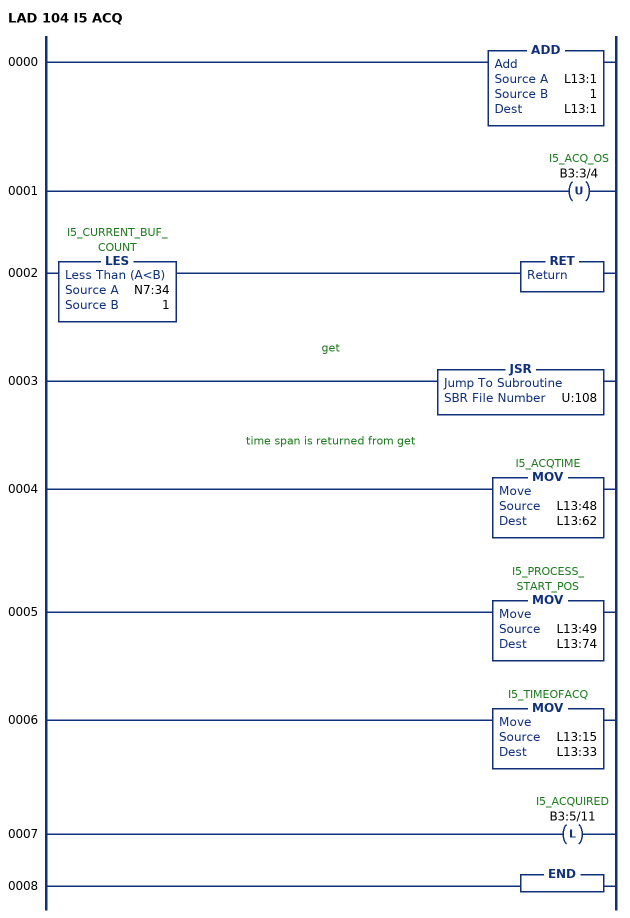
% Rung: 0 %
SOR ADD L13:1 1 L13:1 EOR
% Rung: 1 %
SOR OTU B3:3/4 EOR
%   B3:3/4  I5_ACQ_OS %
% Rung: 2 %
SOR LES N7:34 1 RET EOR
%   N7:34  I5_CURRENT_BUF_COUNT %
% Rung: 3 %
% get %
SOR JSR U:108 EOR
% Rung: 4 %
% time span is returned from get %
SOR MOV L13:48 L13:62 EOR
%   L13:48  I5_TIME_SPAN %
%   L13:62  I5_ACQTIME %
% Rung: 5 %
SOR MOV L13:49 L13:74 EOR
%   L13:49  I5_PULLED_POSITION %
%   L13:74  I5_PROCESS_START_POS %
% Rung: 6 %
SOR MOV L13:15 L13:33 EOR
%   L13:15  THE_TIME %
%   L13:33  I5_TIMEOFACQ %
% Rung: 7 %
SOR OTL B3:5/11 EOR
%   B3:5/11  I5_ACQUIRED %
% Rung: 8 %
SOR END EOR

LADDER 105 "I5 TESTER"
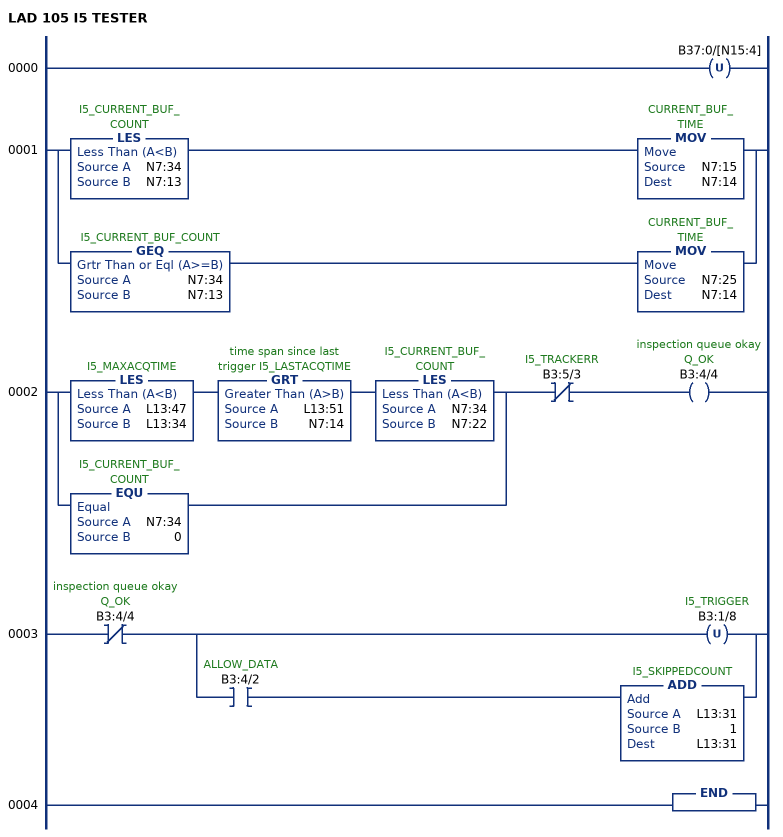
% Rung: 0 %
SOR OTU B37:0/[N15:4] EOR
%   B37:0  TOPGOOD1 %
%   N15:4  I5_TRIG_LOC %
% Rung: 1 %
SOR BST LES N7:34 N7:13 MOV N7:15 N7:14 NXB GEQ N7:34 N7:13 MOV N7:25 N7:14 BND EOR
%   N7:34  I5_CURRENT_BUF_COUNT %
%   N7:13  BUF_TRANS  "cam to pc buf transition" %
%   N7:15  CAM_BUF_TIME  "cam buf time" %
%   N7:14  CURRENT_BUF_TIME %
%   N7:25  PC_BUF_TIME  "pc buf time" %
% Rung: 2 %
SOR BST LES L13:47 L13:34 GRT L13:51 N7:14 LES N7:34 N7:22 NXB EQU N7:34 0 BND XIO B3:5/3 OTE B3:4/4 EOR
%   L13:47  I5_MAXACQTIME %
%   L13:34  MAX_ACQ_ALL  "absolute max acquire time before bypass trigger" %
%   L13:51  I5_LASTACQTIME  "time span since last trigger" %
%   N7:14  CURRENT_BUF_TIME %
%   N7:34  I5_CURRENT_BUF_COUNT %
%   N7:22  MAX_BUF_ALL  "max buffer count alowed before bypass" %
%   B3:5/3  I5_TRACKERR %
%   B3:4/4  Q_OK  "inspection queue okay" %
% Rung: 3 %
SOR XIO B3:4/4 BST OTU B3:1/8 NXB XIC B3:4/2 ADD L13:31 1 L13:31 BND EOR
%   B3:4/4  Q_OK  "inspection queue okay" %
%   B3:1/8  I5_TRIGGER %
%   B3:4/2  ALLOW_DATA %
%   L13:31  I5_SKIPPEDCOUNT %
% Rung: 4 %
SOR END EOR

LADDER 106 "I5 TRIG"
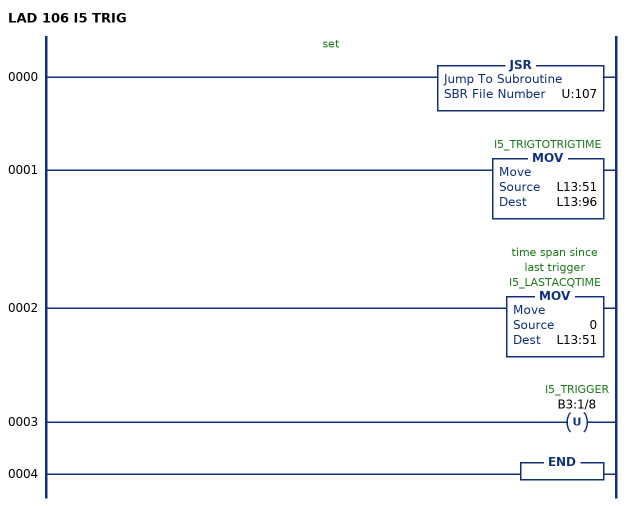
% Rung: 0 %
% set %
SOR JSR U:107 EOR
% Rung: 1 %
SOR MOV L13:51 L13:96 EOR
%   L13:51  I5_LASTACQTIME  "time span since last trigger" %
%   L13:96  I5_TRIGTOTRIGTIME %
% Rung: 2 %
SOR MOV 0 L13:51 EOR
%   L13:51  I5_LASTACQTIME  "time span since last trigger" %
% Rung: 3 %
SOR OTU B3:1/8 EOR
%   B3:1/8  I5_TRIGGER %
% Rung: 4 %
SOR END EOR

LADDER 107 "I5 FIFOSET"
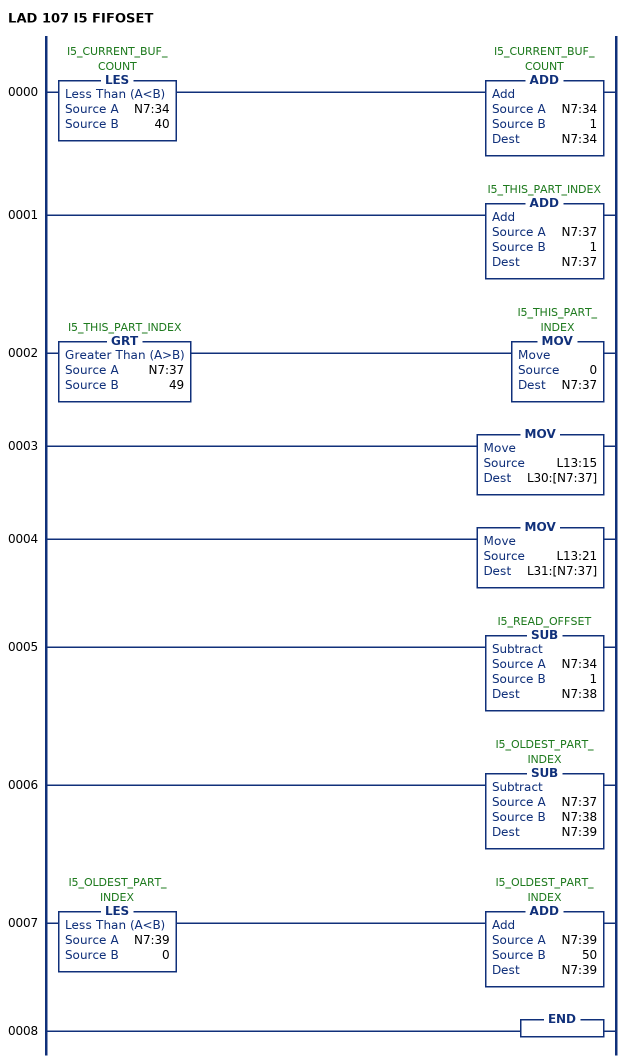
% Rung: 0 %
SOR LES N7:34 40 ADD N7:34 1 N7:34 EOR
%   N7:34  I5_CURRENT_BUF_COUNT %
% Rung: 1 %
SOR ADD N7:37 1 N7:37 EOR
%   N7:37  I5_THIS_PART_INDEX %
% Rung: 2 %
SOR GRT N7:37 49 MOV 0 N7:37 EOR
%   N7:37  I5_THIS_PART_INDEX %
% Rung: 3 %
SOR MOV L13:15 L30:[N7:37] EOR
%   L13:15  THE_TIME %
%   N7:37  I5_THIS_PART_INDEX %
% Rung: 4 %
SOR MOV L13:21 L31:[N7:37] EOR
%   L13:21  TOP_POSITION %
%   N7:37  I5_THIS_PART_INDEX %
% Rung: 5 %
SOR SUB N7:34 1 N7:38 EOR
%   N7:34  I5_CURRENT_BUF_COUNT %
%   N7:38  I5_READ_OFFSET %
% Rung: 6 %
SOR SUB N7:37 N7:38 N7:39 EOR
%   N7:37  I5_THIS_PART_INDEX %
%   N7:38  I5_READ_OFFSET %
%   N7:39  I5_OLDEST_PART_INDEX %
% Rung: 7 %
SOR LES N7:39 0 ADD N7:39 50 N7:39 EOR
%   N7:39  I5_OLDEST_PART_INDEX %
% Rung: 8 %
SOR END EOR

LADDER 108 "I5 FIFOGET"
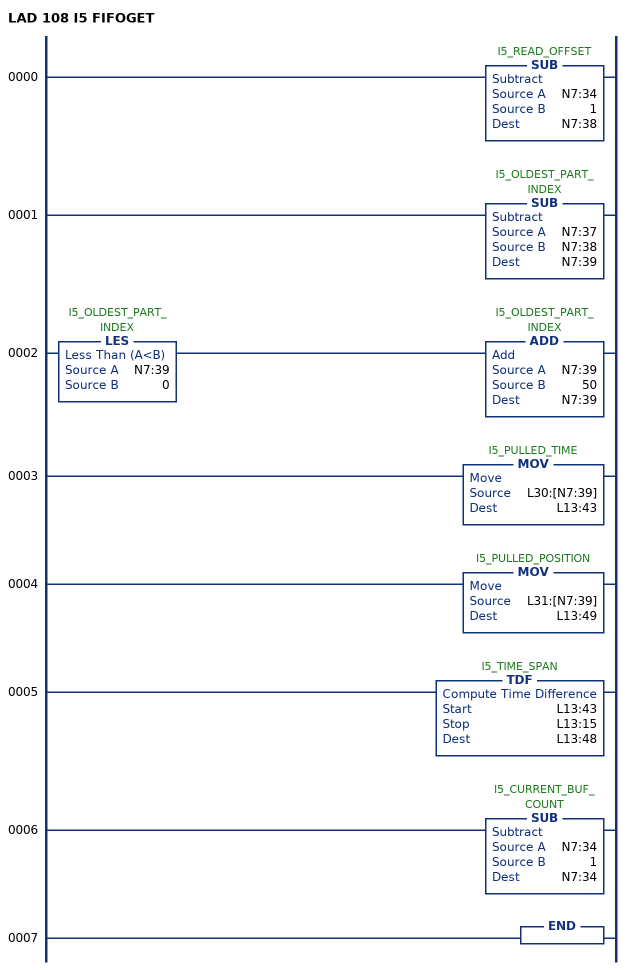
% Rung: 0 %
SOR SUB N7:34 1 N7:38 EOR
%   N7:34  I5_CURRENT_BUF_COUNT %
%   N7:38  I5_READ_OFFSET %
% Rung: 1 %
SOR SUB N7:37 N7:38 N7:39 EOR
%   N7:37  I5_THIS_PART_INDEX %
%   N7:38  I5_READ_OFFSET %
%   N7:39  I5_OLDEST_PART_INDEX %
% Rung: 2 %
SOR LES N7:39 0 ADD N7:39 50 N7:39 EOR
%   N7:39  I5_OLDEST_PART_INDEX %
% Rung: 3 %
SOR MOV L30:[N7:39] L13:43 EOR
%   N7:39  I5_OLDEST_PART_INDEX %
%   L13:43  I5_PULLED_TIME %
% Rung: 4 %
SOR MOV L31:[N7:39] L13:49 EOR
%   N7:39  I5_OLDEST_PART_INDEX %
%   L13:49  I5_PULLED_POSITION %
% Rung: 5 %
SOR TDF L13:43 L13:15 L13:48 EOR
%   L13:43  I5_PULLED_TIME %
%   L13:15  THE_TIME %
%   L13:48  I5_TIME_SPAN %
% Rung: 6 %
SOR SUB N7:34 1 N7:34 EOR
%   N7:34  I5_CURRENT_BUF_COUNT %
% Rung: 7 %
SOR END EOR

LADDER 109 "I5 DATA"
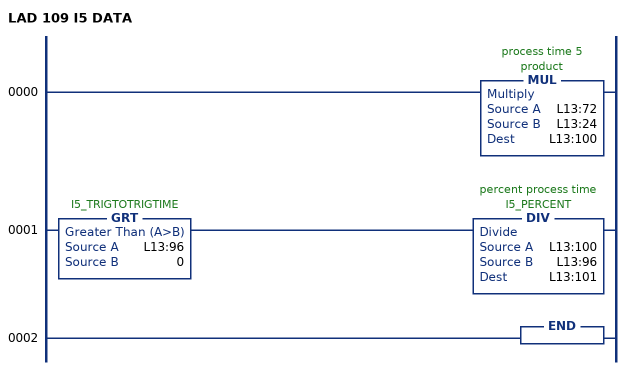
% Rung: 0 %
SOR MUL L13:72 L13:24 L13:100 EOR
%   L13:72  I5_PROCESSTIME %
%   L13:24  "multiplyer to make devision come out to a percentage" %
%   L13:100  "process time 5 product" %
% Rung: 1 %
SOR GRT L13:96 0 DIV L13:100 L13:96 L13:101 EOR
%   L13:96  I5_TRIGTOTRIGTIME %
%   L13:100  "process time 5 product" %
%   L13:101  I5_PERCENT  "percent process time" %
% Rung: 2 %
SOR END EOR

LADDER 110 "I5 FAULT"
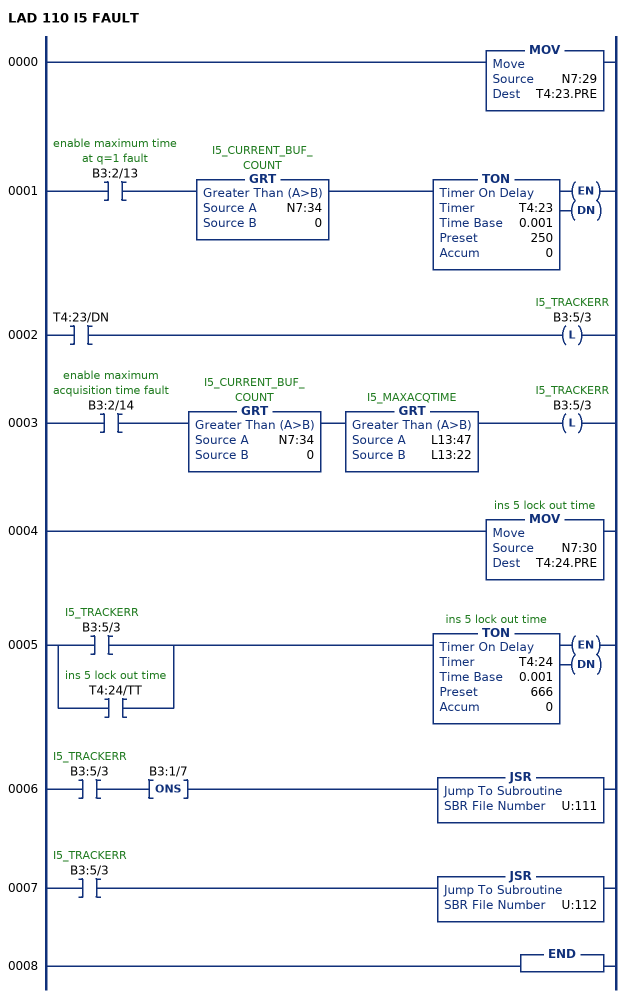
% Rung: 0 %
SOR MOV N7:29 T4:23.PRE EOR
%   N7:29  "max allowed ms time for q to be above 1 if safe fault is used" %
% Rung: 1 %
SOR XIC B3:2/13 GRT N7:34 0 TON T4:23 0.001 250 0 EOR
%   B3:2/13  "enable maximum time at q=1 fault" %
%   N7:34  I5_CURRENT_BUF_COUNT %
% Rung: 2 %
SOR XIC T4:23/DN OTL B3:5/3 EOR
%   B3:5/3  I5_TRACKERR %
% Rung: 3 %
SOR XIC B3:2/14 GRT N7:34 0 GRT L13:47 L13:22 OTL B3:5/3 EOR
%   B3:2/14  "enable maximum acquisition time fault" %
%   N7:34  I5_CURRENT_BUF_COUNT %
%   L13:47  I5_MAXACQTIME %
%   L13:22  "maximum of the longest acquire time allowed if maximum acquire time fault is enabled" %
%   B3:5/3  I5_TRACKERR %
% Rung: 4 %
SOR MOV N7:30 T4:24.PRE EOR
%   N7:30  "ms time setting to lock out inspection to give all pending images a chance to clear" %
%   T4:24  "ins 5 lock out time" %
% Rung: 5 %
SOR BST XIC B3:5/3 NXB XIC T4:24/TT BND TON T4:24 0.001 666 0 EOR
%   B3:5/3  I5_TRACKERR %
%   T4:24  "ins 5 lock out time" %
% Rung: 6 %
SOR XIC B3:5/3 ONS B3:1/7 JSR U:111 EOR
%   B3:5/3  I5_TRACKERR %
% Rung: 7 %
SOR XIC B3:5/3 JSR U:112 EOR
%   B3:5/3  I5_TRACKERR %
% Rung: 8 %
SOR END EOR

LADDER 111 "I5 FIX1"
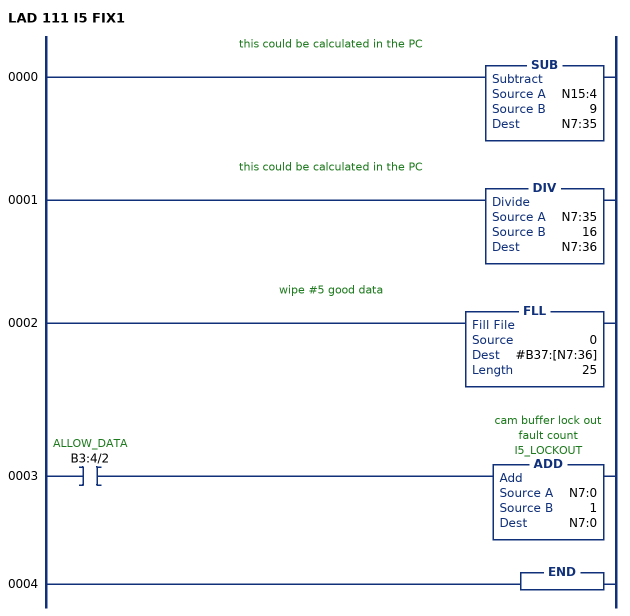
% Rung: 0 %
% this could be calculated in the PC %
SOR SUB N15:4 9 N7:35 EOR
%   N15:4  I5_TRIG_LOC %
% Rung: 1 %
% this could be calculated in the PC %
SOR DIV N7:35 16 N7:36 EOR
% Rung: 2 %
% wipe #5 good data %
SOR FLL 0 #B37:[N7:36] 25 EOR
% Rung: 3 %
SOR XIC B3:4/2 ADD N7:0 1 N7:0 EOR
%   B3:4/2  ALLOW_DATA %
%   N7:0  I5_LOCKOUT  "cam buffer lock out fault count" %
% Rung: 4 %
SOR END EOR

LADDER 112 "I5 FIX2"
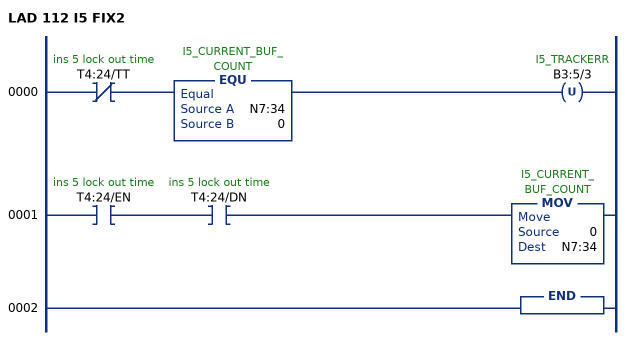
% Rung: 0 %
SOR XIO T4:24/TT EQU N7:34 0 OTU B3:5/3 EOR
%   T4:24  "ins 5 lock out time" %
%   N7:34  I5_CURRENT_BUF_COUNT %
%   B3:5/3  I5_TRACKERR %
% Rung: 1 %
SOR XIC T4:24/EN XIC T4:24/DN MOV 0 N7:34 EOR
%   T4:24  "ins 5 lock out time" %
%   N7:34  I5_CURRENT_BUF_COUNT %
% Rung: 2 %
SOR END EOR

LADDER 120 "I6"
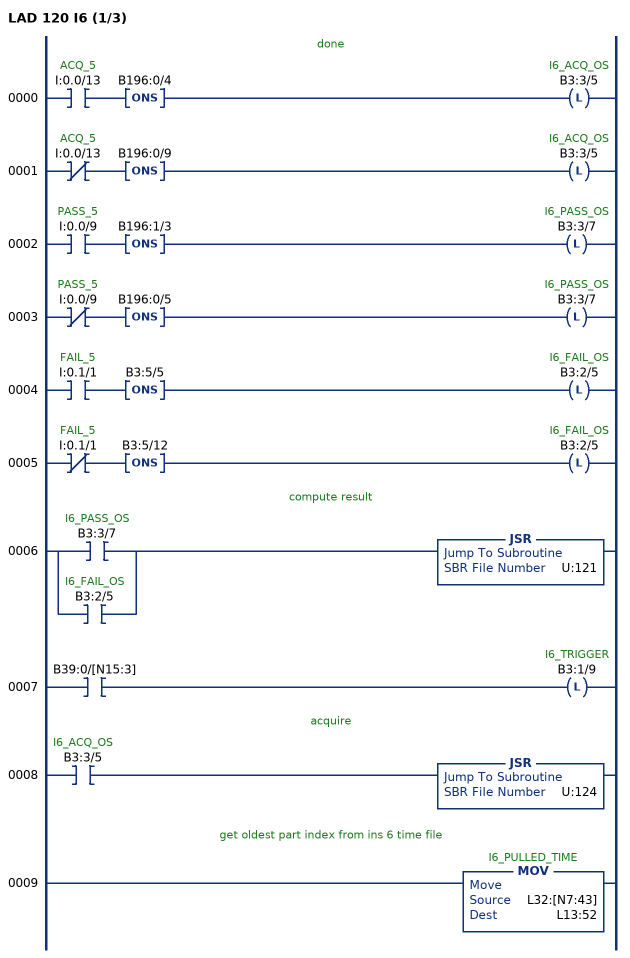
% Rung: 0 %
% done %
SOR XIC I:0.0/13 ONS B196:0/4 OTL B3:3/5 EOR
%   I:0.0/13  ACQ_5 %
%   B3:3/5  I6_ACQ_OS %
% Rung: 1 %
SOR XIO I:0.0/13 ONS B196:0/9 OTL B3:3/5 EOR
%   I:0.0/13  ACQ_5 %
%   B3:3/5  I6_ACQ_OS %
% Rung: 2 %
SOR XIC I:0.0/9 ONS B196:1/3 OTL B3:3/7 EOR
%   I:0.0/9  PASS_5 %
%   B3:3/7  I6_PASS_OS %
% Rung: 3 %
SOR XIO I:0.0/9 ONS B196:0/5 OTL B3:3/7 EOR
%   I:0.0/9  PASS_5 %
%   B3:3/7  I6_PASS_OS %
% Rung: 4 %
SOR XIC I:0.1/1 ONS B3:5/5 OTL B3:2/5 EOR
%   I:0.1/1  FAIL_5 %
%   B3:2/5  I6_FAIL_OS %
% Rung: 5 %
SOR XIO I:0.1/1 ONS B3:5/12 OTL B3:2/5 EOR
%   I:0.1/1  FAIL_5 %
%   B3:2/5  I6_FAIL_OS %
% Rung: 6 %
% compute result %
SOR BST XIC B3:3/7 NXB XIC B3:2/5 BND JSR U:121 EOR
%   B3:3/7  I6_PASS_OS %
%   B3:2/5  I6_FAIL_OS %
% Rung: 7 %
SOR XIC B39:0/[N15:3] OTL B3:1/9 EOR
%   B39:0  TOPGOOD2 %
%   N15:3  I6_TRIG_LOC %
%   B3:1/9  I6_TRIGGER %
% Rung: 8 %
% acquire %
SOR XIC B3:3/5 JSR U:124 EOR
%   B3:3/5  I6_ACQ_OS %
% Rung: 9 %
% get oldest part index from ins 6 time file %
SOR MOV L32:[N7:43] L13:52 EOR
%   N7:43  I6_OLDEST_PART_INDEX %
%   L13:52  I6_PULLED_TIME %

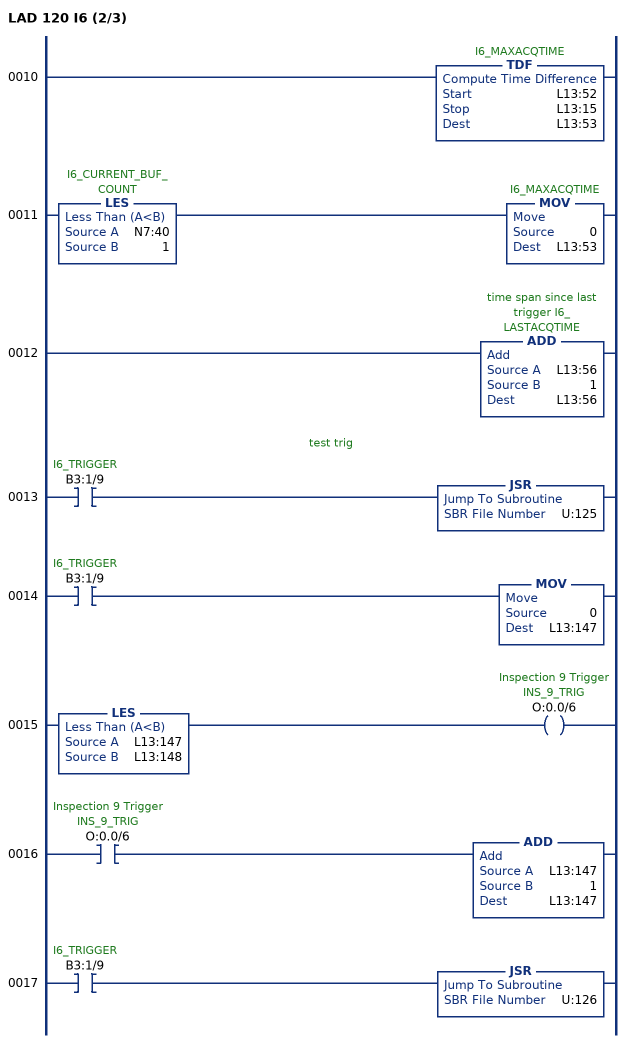
% Rung: 10 %
SOR TDF L13:52 L13:15 L13:53 EOR
%   L13:52  I6_PULLED_TIME %
%   L13:15  THE_TIME %
%   L13:53  I6_MAXACQTIME %
% Rung: 11 %
SOR LES N7:40 1 MOV 0 L13:53 EOR
%   N7:40  I6_CURRENT_BUF_COUNT %
%   L13:53  I6_MAXACQTIME %
% Rung: 12 %
SOR ADD L13:56 1 L13:56 EOR
%   L13:56  I6_LASTACQTIME  "time span since last trigger" %
% Rung: 13 %
% test trig %
SOR XIC B3:1/9 JSR U:125 EOR
%   B3:1/9  I6_TRIGGER %
% Rung: 14 %
SOR XIC B3:1/9 MOV 0 L13:147 EOR
%   B3:1/9  I6_TRIGGER %
% Rung: 15 %
SOR LES L13:147 L13:148 OTE O:0.0/6 EOR
%   O:0.0/6  INS_9_TRIG  "Inspection 9 Trigger" %
% Rung: 16 %
SOR XIC O:0.0/6 ADD L13:147 1 L13:147 EOR
%   O:0.0/6  INS_9_TRIG  "Inspection 9 Trigger" %
% Rung: 17 %
SOR XIC B3:1/9 JSR U:126 EOR
%   B3:1/9  I6_TRIGGER %

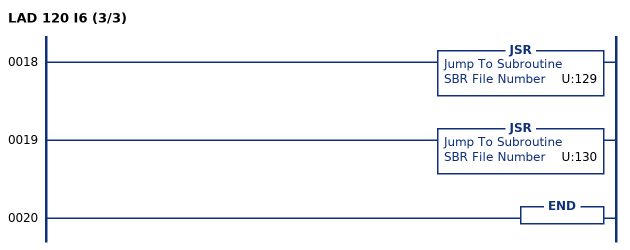
% Rung: 18 %
SOR JSR U:129 EOR
% Rung: 19 %
SOR JSR U:130 EOR
% Rung: 20 %
SOR END EOR

LADDER 121 "I6 RESULT"
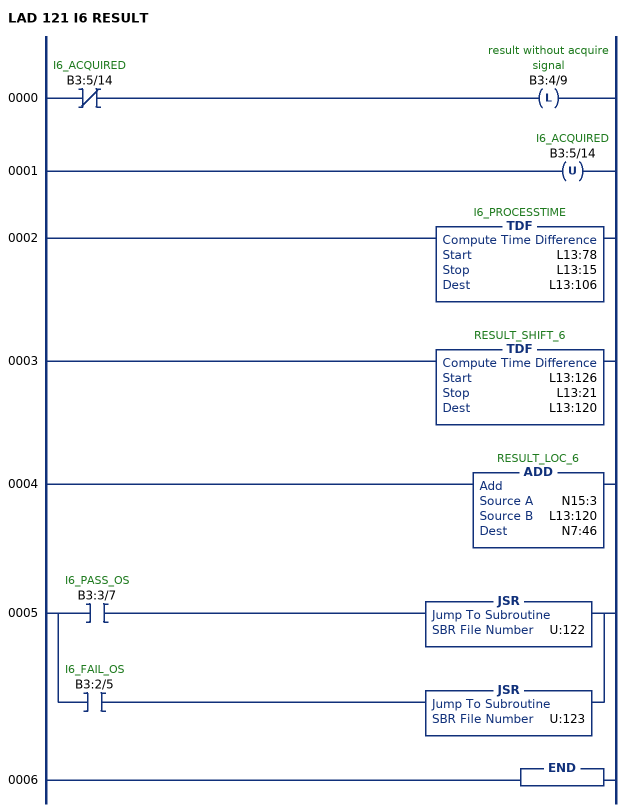
% Rung: 0 %
SOR XIO B3:5/14 OTL B3:4/9 EOR
%   B3:5/14  I6_ACQUIRED %
%   B3:4/9  "result without acquire signal" %
% Rung: 1 %
SOR OTU B3:5/14 EOR
%   B3:5/14  I6_ACQUIRED %
% Rung: 2 %
SOR TDF L13:78 L13:15 L13:106 EOR
%   L13:78  I6_TIMEOFACQ %
%   L13:15  THE_TIME %
%   L13:106  I6_PROCESSTIME %
% Rung: 3 %
SOR TDF L13:126 L13:21 L13:120 EOR
%   L13:126  I6_PROCESS_START_POS %
%   L13:21  TOP_POSITION %
%   L13:120  RESULT_SHIFT_6 %
% Rung: 4 %
SOR ADD N15:3 L13:120 N7:46 EOR
%   N15:3  I6_TRIG_LOC %
%   L13:120  RESULT_SHIFT_6 %
%   N7:46  RESULT_LOC_6 %
% Rung: 5 %
SOR BST XIC B3:3/7 JSR U:122 NXB XIC B3:2/5 JSR U:123 BND EOR
%   B3:3/7  I6_PASS_OS %
%   B3:2/5  I6_FAIL_OS %
% Rung: 6 %
SOR END EOR

LADDER 122 "I6 PASS"
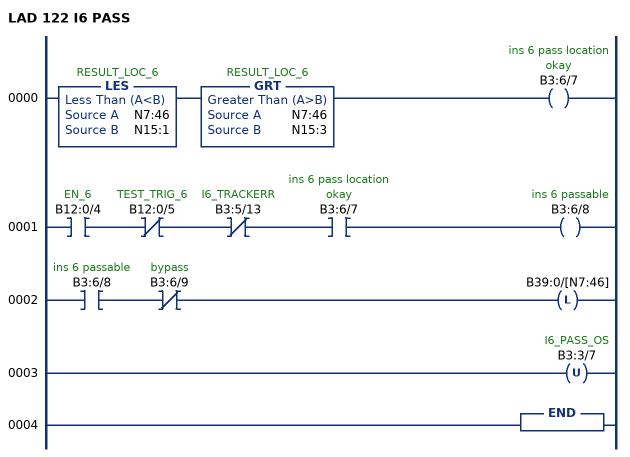
% Rung: 0 %
SOR LES N7:46 N15:1 GRT N7:46 N15:3 OTE B3:6/7 EOR
%   N7:46  RESULT_LOC_6 %
%   N15:1  I8_TRIG_LOC %
%   N15:3  I6_TRIG_LOC %
%   B3:6/7  "ins 6 pass location okay" %
% Rung: 1 %
SOR XIC B12:0/4 XIO B12:0/5 XIO B3:5/13 XIC B3:6/7 OTE B3:6/8 EOR
%   B12:0/4  EN_6 %
%   B12:0/5  TEST_TRIG_6 %
%   B3:5/13  I6_TRACKERR %
%   B3:6/7  "ins 6 pass location okay" %
%   B3:6/8  "ins 6 passable" %
% Rung: 2 %
SOR XIC B3:6/8 XIO B3:6/9 OTL B39:0/[N7:46] EOR
%   B3:6/8  "ins 6 passable" %
%   B3:6/9  "bypass" %
%   B39:0  TOPGOOD2 %
%   N7:46  RESULT_LOC_6 %
% Rung: 3 %
SOR OTU B3:3/7 EOR
%   B3:3/7  I6_PASS_OS %
% Rung: 4 %
SOR END EOR

LADDER 123 "I6 FAIL"
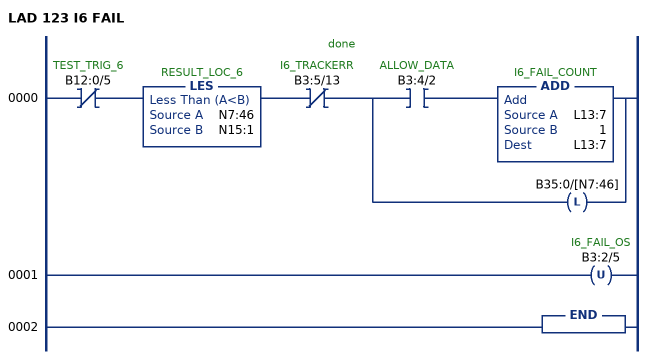
% Rung: 0 %
% done %
SOR XIO B12:0/5 LES N7:46 N15:1 XIO B3:5/13 BST XIC B3:4/2 ADD L13:7 1 L13:7 NXB OTL B35:0/[N7:46] BND EOR
%   B12:0/5  TEST_TRIG_6 %
%   N7:46  RESULT_LOC_6 %
%   N15:1  I8_TRIG_LOC %
%   B3:5/13  I6_TRACKERR %
%   B3:4/2  ALLOW_DATA %
%   L13:7  I6_FAIL_COUNT %
%   B35:0  TOP_NG %
% Rung: 1 %
SOR OTU B3:2/5 EOR
%   B3:2/5  I6_FAIL_OS %
% Rung: 2 %
SOR END EOR

LADDER 124 "I6 ACQ"
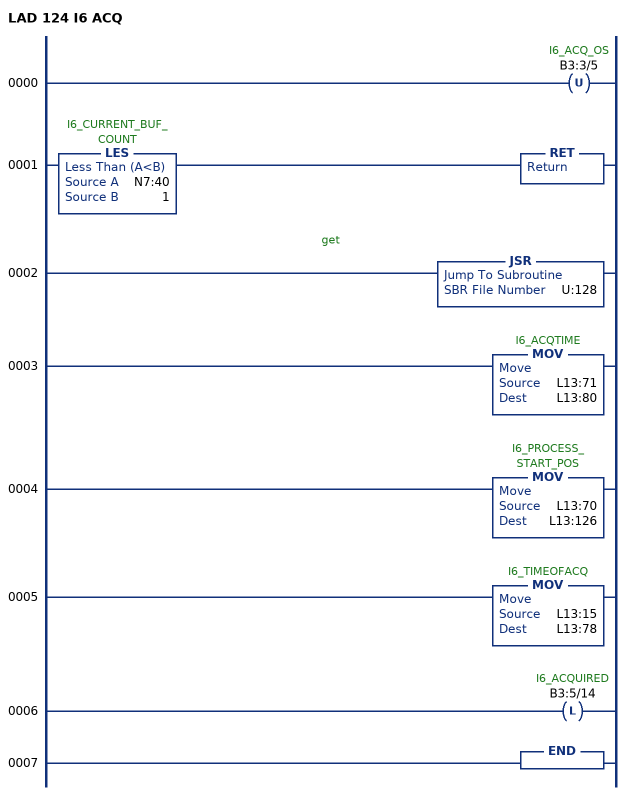
% Rung: 0 %
SOR OTU B3:3/5 EOR
%   B3:3/5  I6_ACQ_OS %
% Rung: 1 %
SOR LES N7:40 1 RET EOR
%   N7:40  I6_CURRENT_BUF_COUNT %
% Rung: 2 %
% get %
SOR JSR U:128 EOR
% Rung: 3 %
SOR MOV L13:71 L13:80 EOR
%   L13:71  I6_TIME_SPAN %
%   L13:80  I6_ACQTIME %
% Rung: 4 %
SOR MOV L13:70 L13:126 EOR
%   L13:70  I6_PULLED_POSITION %
%   L13:126  I6_PROCESS_START_POS %
% Rung: 5 %
SOR MOV L13:15 L13:78 EOR
%   L13:15  THE_TIME %
%   L13:78  I6_TIMEOFACQ %
% Rung: 6 %
SOR OTL B3:5/14 EOR
%   B3:5/14  I6_ACQUIRED %
% Rung: 7 %
SOR END EOR

LADDER 125 "I6 TESTER"
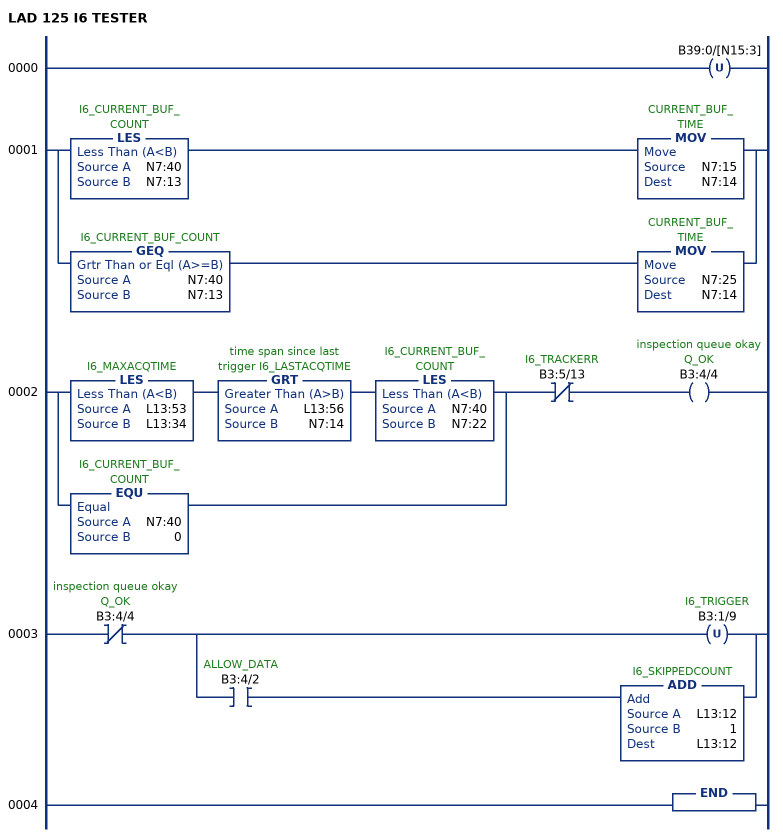
% Rung: 0 %
SOR OTU B39:0/[N15:3] EOR
%   B39:0  TOPGOOD2 %
%   N15:3  I6_TRIG_LOC %
% Rung: 1 %
SOR BST LES N7:40 N7:13 MOV N7:15 N7:14 NXB GEQ N7:40 N7:13 MOV N7:25 N7:14 BND EOR
%   N7:40  I6_CURRENT_BUF_COUNT %
%   N7:13  BUF_TRANS  "cam to pc buf transition" %
%   N7:15  CAM_BUF_TIME  "cam buf time" %
%   N7:14  CURRENT_BUF_TIME %
%   N7:25  PC_BUF_TIME  "pc buf time" %
% Rung: 2 %
SOR BST LES L13:53 L13:34 GRT L13:56 N7:14 LES N7:40 N7:22 NXB EQU N7:40 0 BND XIO B3:5/13 OTE B3:4/4 EOR
%   L13:53  I6_MAXACQTIME %
%   L13:34  MAX_ACQ_ALL  "absolute max acquire time before bypass trigger" %
%   L13:56  I6_LASTACQTIME  "time span since last trigger" %
%   N7:14  CURRENT_BUF_TIME %
%   N7:40  I6_CURRENT_BUF_COUNT %
%   N7:22  MAX_BUF_ALL  "max buffer count alowed before bypass" %
%   B3:5/13  I6_TRACKERR %
%   B3:4/4  Q_OK  "inspection queue okay" %
% Rung: 3 %
SOR XIO B3:4/4 BST OTU B3:1/9 NXB XIC B3:4/2 ADD L13:12 1 L13:12 BND EOR
%   B3:4/4  Q_OK  "inspection queue okay" %
%   B3:1/9  I6_TRIGGER %
%   B3:4/2  ALLOW_DATA %
%   L13:12  I6_SKIPPEDCOUNT %
% Rung: 4 %
SOR END EOR

LADDER 126 "I6 TRIG"
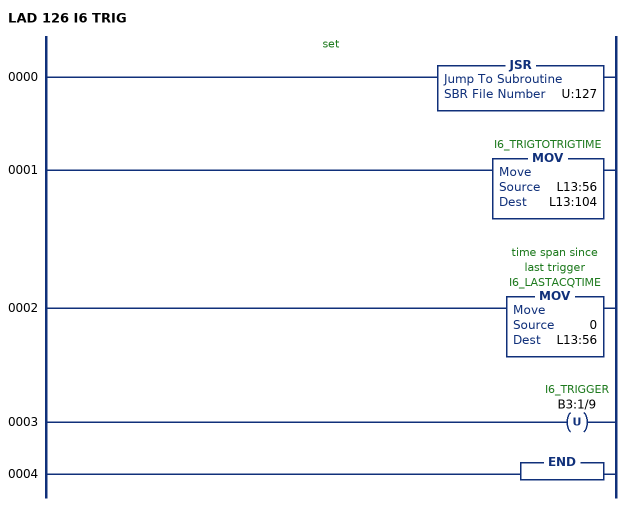
% Rung: 0 %
% set %
SOR JSR U:127 EOR
% Rung: 1 %
SOR MOV L13:56 L13:104 EOR
%   L13:56  I6_LASTACQTIME  "time span since last trigger" %
%   L13:104  I6_TRIGTOTRIGTIME %
% Rung: 2 %
SOR MOV 0 L13:56 EOR
%   L13:56  I6_LASTACQTIME  "time span since last trigger" %
% Rung: 3 %
SOR OTU B3:1/9 EOR
%   B3:1/9  I6_TRIGGER %
% Rung: 4 %
SOR END EOR

LADDER 127 "I6 FIFOSET"
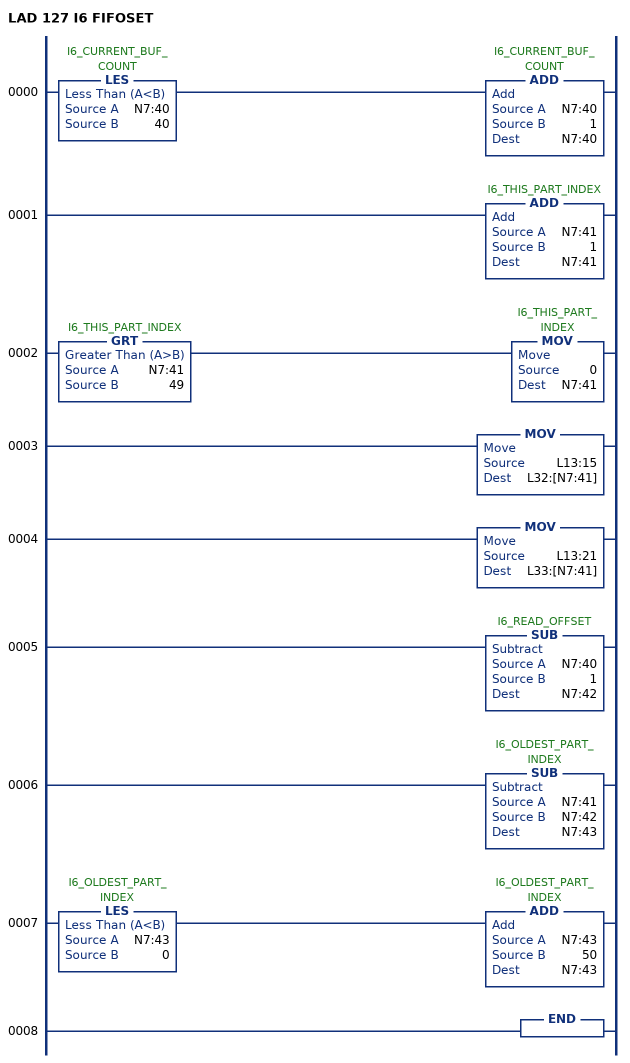
% Rung: 0 %
SOR LES N7:40 40 ADD N7:40 1 N7:40 EOR
%   N7:40  I6_CURRENT_BUF_COUNT %
% Rung: 1 %
SOR ADD N7:41 1 N7:41 EOR
%   N7:41  I6_THIS_PART_INDEX %
% Rung: 2 %
SOR GRT N7:41 49 MOV 0 N7:41 EOR
%   N7:41  I6_THIS_PART_INDEX %
% Rung: 3 %
SOR MOV L13:15 L32:[N7:41] EOR
%   L13:15  THE_TIME %
%   N7:41  I6_THIS_PART_INDEX %
% Rung: 4 %
SOR MOV L13:21 L33:[N7:41] EOR
%   L13:21  TOP_POSITION %
%   N7:41  I6_THIS_PART_INDEX %
% Rung: 5 %
SOR SUB N7:40 1 N7:42 EOR
%   N7:40  I6_CURRENT_BUF_COUNT %
%   N7:42  I6_READ_OFFSET %
% Rung: 6 %
SOR SUB N7:41 N7:42 N7:43 EOR
%   N7:41  I6_THIS_PART_INDEX %
%   N7:42  I6_READ_OFFSET %
%   N7:43  I6_OLDEST_PART_INDEX %
% Rung: 7 %
SOR LES N7:43 0 ADD N7:43 50 N7:43 EOR
%   N7:43  I6_OLDEST_PART_INDEX %
% Rung: 8 %
SOR END EOR

LADDER 128 "I6 FIFOGET"
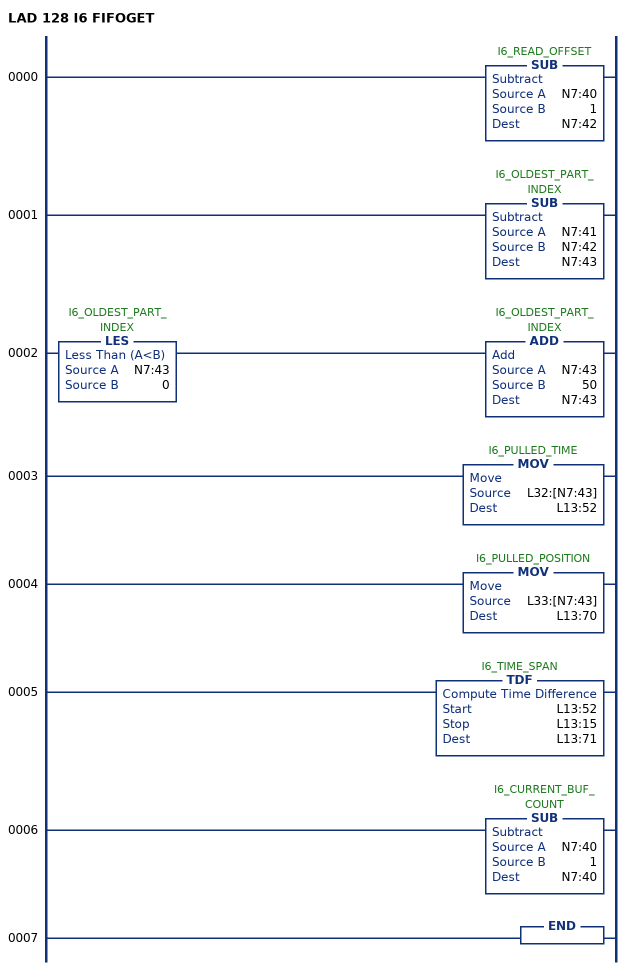
% Rung: 0 %
SOR SUB N7:40 1 N7:42 EOR
%   N7:40  I6_CURRENT_BUF_COUNT %
%   N7:42  I6_READ_OFFSET %
% Rung: 1 %
SOR SUB N7:41 N7:42 N7:43 EOR
%   N7:41  I6_THIS_PART_INDEX %
%   N7:42  I6_READ_OFFSET %
%   N7:43  I6_OLDEST_PART_INDEX %
% Rung: 2 %
SOR LES N7:43 0 ADD N7:43 50 N7:43 EOR
%   N7:43  I6_OLDEST_PART_INDEX %
% Rung: 3 %
SOR MOV L32:[N7:43] L13:52 EOR
%   N7:43  I6_OLDEST_PART_INDEX %
%   L13:52  I6_PULLED_TIME %
% Rung: 4 %
SOR MOV L33:[N7:43] L13:70 EOR
%   N7:43  I6_OLDEST_PART_INDEX %
%   L13:70  I6_PULLED_POSITION %
% Rung: 5 %
SOR TDF L13:52 L13:15 L13:71 EOR
%   L13:52  I6_PULLED_TIME %
%   L13:15  THE_TIME %
%   L13:71  I6_TIME_SPAN %
% Rung: 6 %
SOR SUB N7:40 1 N7:40 EOR
%   N7:40  I6_CURRENT_BUF_COUNT %
% Rung: 7 %
SOR END EOR

LADDER 129 "I6 DATA"
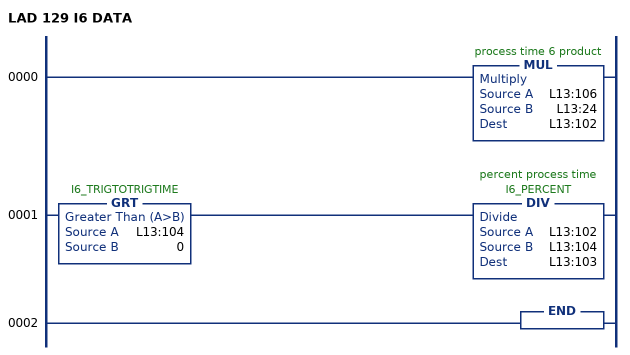
% Rung: 0 %
SOR MUL L13:106 L13:24 L13:102 EOR
%   L13:106  I6_PROCESSTIME %
%   L13:24  "multiplyer to make devision come out to a percentage" %
%   L13:102  "process time 6 product" %
% Rung: 1 %
SOR GRT L13:104 0 DIV L13:102 L13:104 L13:103 EOR
%   L13:104  I6_TRIGTOTRIGTIME %
%   L13:102  "process time 6 product" %
%   L13:103  I6_PERCENT  "percent process time" %
% Rung: 2 %
SOR END EOR

LADDER 130 "I6 FAULT"
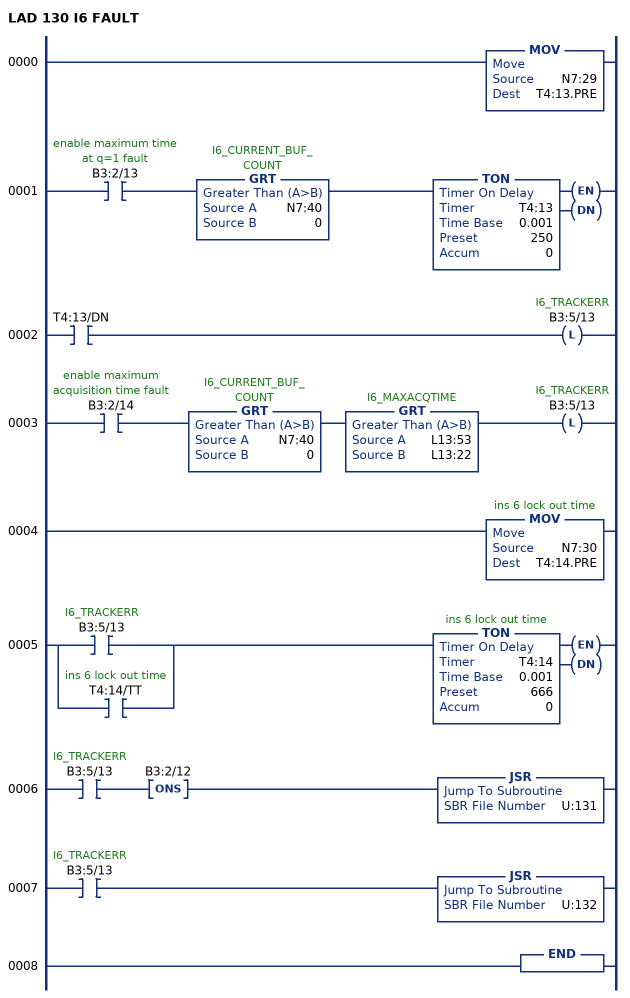
% Rung: 0 %
SOR MOV N7:29 T4:13.PRE EOR
%   N7:29  "max allowed ms time for q to be above 1 if safe fault is used" %
% Rung: 1 %
SOR XIC B3:2/13 GRT N7:40 0 TON T4:13 0.001 250 0 EOR
%   B3:2/13  "enable maximum time at q=1 fault" %
%   N7:40  I6_CURRENT_BUF_COUNT %
% Rung: 2 %
SOR XIC T4:13/DN OTL B3:5/13 EOR
%   B3:5/13  I6_TRACKERR %
% Rung: 3 %
SOR XIC B3:2/14 GRT N7:40 0 GRT L13:53 L13:22 OTL B3:5/13 EOR
%   B3:2/14  "enable maximum acquisition time fault" %
%   N7:40  I6_CURRENT_BUF_COUNT %
%   L13:53  I6_MAXACQTIME %
%   L13:22  "maximum of the longest acquire time allowed if maximum acquire time fault is enabled" %
%   B3:5/13  I6_TRACKERR %
% Rung: 4 %
SOR MOV N7:30 T4:14.PRE EOR
%   N7:30  "ms time setting to lock out inspection to give all pending images a chance to clear" %
%   T4:14  "ins 6 lock out time" %
% Rung: 5 %
SOR BST XIC B3:5/13 NXB XIC T4:14/TT BND TON T4:14 0.001 666 0 EOR
%   B3:5/13  I6_TRACKERR %
%   T4:14  "ins 6 lock out time" %
% Rung: 6 %
SOR XIC B3:5/13 ONS B3:2/12 JSR U:131 EOR
%   B3:5/13  I6_TRACKERR %
% Rung: 7 %
SOR XIC B3:5/13 JSR U:132 EOR
%   B3:5/13  I6_TRACKERR %
% Rung: 8 %
SOR END EOR

LADDER 131 "I6 FIX1"
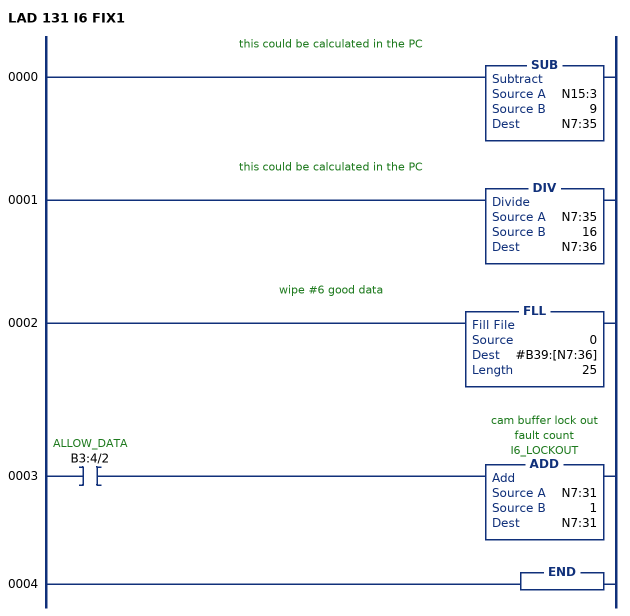
% Rung: 0 %
% this could be calculated in the PC %
SOR SUB N15:3 9 N7:35 EOR
%   N15:3  I6_TRIG_LOC %
% Rung: 1 %
% this could be calculated in the PC %
SOR DIV N7:35 16 N7:36 EOR
% Rung: 2 %
% wipe #6 good data %
SOR FLL 0 #B39:[N7:36] 25 EOR
% Rung: 3 %
SOR XIC B3:4/2 ADD N7:31 1 N7:31 EOR
%   B3:4/2  ALLOW_DATA %
%   N7:31  I6_LOCKOUT  "cam buffer lock out fault count" %
% Rung: 4 %
SOR END EOR

LADDER 132 "I6 FIX2"
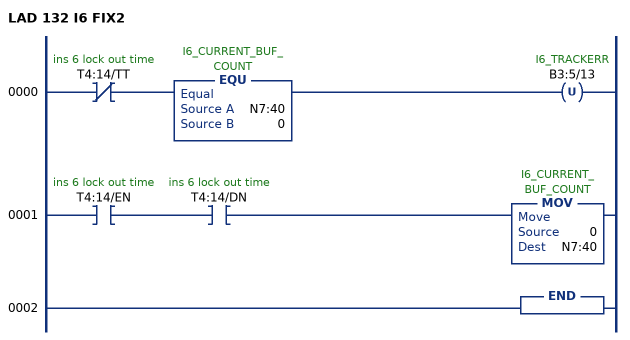
% Rung: 0 %
SOR XIO T4:14/TT EQU N7:40 0 OTU B3:5/13 EOR
%   T4:14  "ins 6 lock out time" %
%   N7:40  I6_CURRENT_BUF_COUNT %
%   B3:5/13  I6_TRACKERR %
% Rung: 1 %
SOR XIC T4:14/EN XIC T4:14/DN MOV 0 N7:40 EOR
%   T4:14  "ins 6 lock out time" %
%   N7:40  I6_CURRENT_BUF_COUNT %
% Rung: 2 %
SOR END EOR

LADDER 140 "I7"
